FUNCTION_BLOCK skPush (* Composite Function Block Type *)
  (* Standard: 61499-2 *)
  (* Version 0.0, 11/8/2025, codex, template *)
  PACKAGE Main;
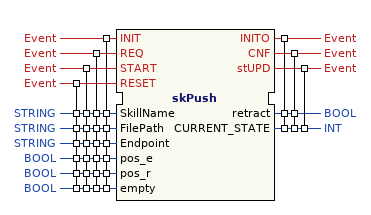
  EVENT_INPUT
    INIT WITH SkillName, FilePath, Endpoint, pos_e, pos_r, empty; (* Initialization Request *)
    REQ WITH SkillName, FilePath, Endpoint, pos_e, pos_r, empty; (* Normal Execution Request *)
    START WITH SkillName, FilePath, Endpoint, pos_e, pos_r, empty;
    RESET WITH SkillName, FilePath, Endpoint, pos_e, pos_r, empty;
  END_EVENT
  EVENT_OUTPUT
    INITO WITH retract, CURRENT_STATE; (* Initialization Confirm *)
    CNF WITH retract, CURRENT_STATE; (* Execution Confirmation *)
    stUPD WITH CURRENT_STATE;
  END_EVENT
  VAR_INPUT
    SkillName : STRING;
    FilePath : STRING;
    Endpoint : STRING;
    pos_e : BOOL; (* Input event qualifier *)
    pos_r : BOOL;
    empty : BOOL;
  END_VAR
  VAR_OUTPUT
    retract : BOOL; (* Output event qualifier *)
    CURRENT_STATE : INT;
  END_VAR
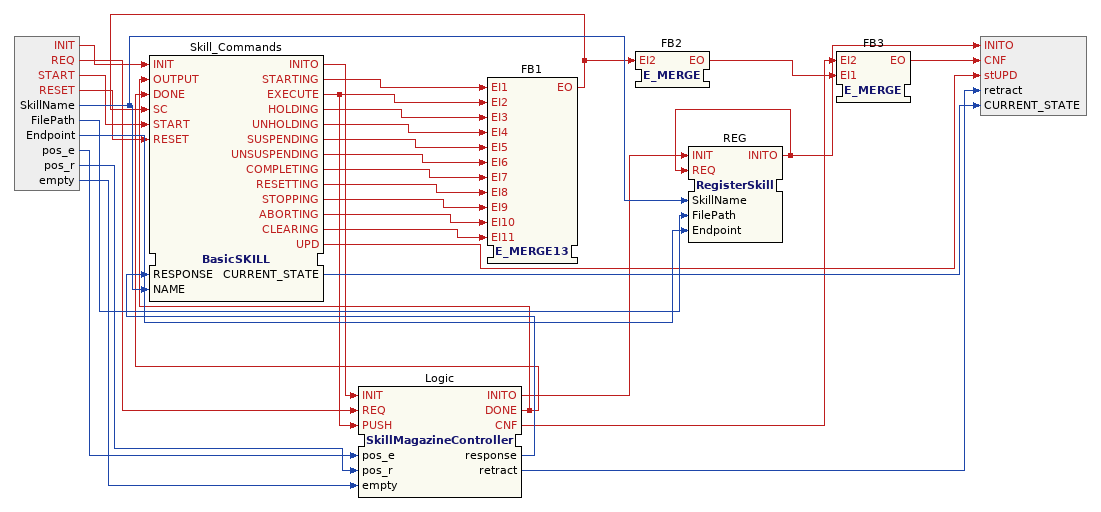
  FBS
    Skill_Commands : BasicSKILL;
    REG : RegisterSkill;
    Logic : SkillMagazineController;
    FB1 : E_MERGE13;
    FB2 : E_MERGE;
    FB3 : E_MERGE;
  END_FBS
  EVENT_CONNECTIONS
    INIT TO Skill_Commands.INIT;
    Skill_Commands.INITO TO Logic.INIT;
    Logic.INITO TO REG.INIT;
    REG.INITO TO REG.REQ;
    REQ TO Logic.REQ;
    REG.INITO TO INITO;
    Skill_Commands.STARTING TO FB1.EI1;
    Skill_Commands.EXECUTE TO Logic.PUSH;
    Skill_Commands.EXECUTE TO FB1.EI2;
    Skill_Commands.HOLDING TO FB1.EI3;
    Skill_Commands.UNHOLDING TO FB1.EI4;
    Skill_Commands.SUSPENDING TO FB1.EI5;
    Skill_Commands.UNSUSPENDING TO FB1.EI6;
    Skill_Commands.COMPLETING TO FB1.EI7;
    Skill_Commands.RESETTING TO FB1.EI8;
    Skill_Commands.STOPPING TO FB1.EI9;
    Skill_Commands.ABORTING TO FB1.EI10;
    Skill_Commands.CLEARING TO FB1.EI11;
    Logic.DONE TO Skill_Commands.OUTPUT;
    Logic.CNF TO FB3.EI2;
    Logic.DONE TO Skill_Commands.DONE;
    FB3.EO TO CNF;
    FB1.EO TO Skill_Commands.SC;
    START TO Skill_Commands.START;
    RESET TO Skill_Commands.RESET;
    FB2.EO TO FB3.EI1;
    FB1.EO TO FB2.EI2;
    Skill_Commands.UPD TO stUPD;
  END_CONNECTIONS
  DATA_CONNECTIONS
    SkillName TO REG.SkillName;
    FilePath TO REG.FilePath;
    Endpoint TO REG.Endpoint;
    Logic.response TO Skill_Commands.RESPONSE;
    pos_e TO Logic.pos_e;
    pos_r TO Logic.pos_r;
    Logic.retract TO retract;
    empty TO Logic.empty;
    SkillName TO Skill_Commands.NAME;
    Skill_Commands.CURRENT_STATE TO CURRENT_STATE;
  END_CONNECTIONS
END_FUNCTION_BLOCK
